{attribute 'qualified_only'}
{attribute 'strict'}
{attribute 'to_string'}
TYPE FILE_MOVE_POINTER_TYPE :
(
	FROM_FILE_BEGINNING,
	FROM_CURRENT_POSITION,
	FROM_FILE_END
);
END_TYPE

(* stored: Version 1.1.0.1
   DUT FILE_MOVE_POINTER_TYPE: Id {07c9d863-df62-4f09-bd47-459f824710a7} *)
